Staubli VAL3: setCenter.pgx

program setCenter()
begin
end
